{attribute 'qualified_only'}
{attribute 'strict'}
{attribute 'to_string'}
TYPE E_LeviState :
(
	LEVI_IDLE := 0,
	LEVI_INIT := 1,
	LEVI_PULLUP := 2,
	LEVI_DROPDOWN := 3,
	LEVI_CONTROL := 4,
	LEVI_ERROR := 5,
	LEVI_DRIVERESET := 6,
	LEVI_SYSTEM_CHECK := 7,
	LEVI_HARD_RESET := 8
	
);
END_TYPE

(* stored: Version 1.1.0.1
   DUT E_LeviState: Id {658b4874-55b1-49b5-9d14-1cfaa576f232} *)
